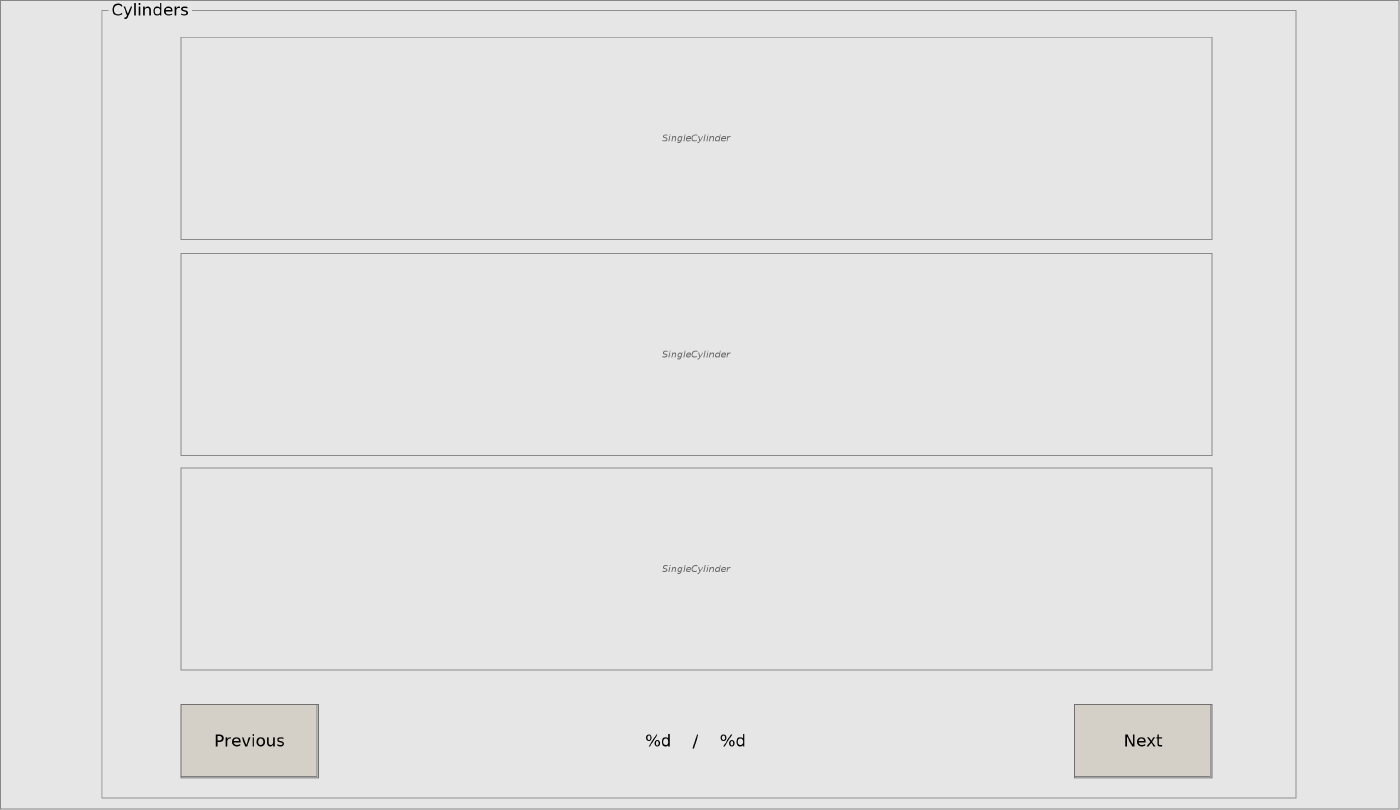
VISUALIZATION PageManualCylinders  // 1520x880
VAR_IN_OUT
	btnPrevious			: BOOL;
	btnNext				: BOOL;
	bPreviousInvisible	: BOOL;
	bNextInvisible		: BOOL;
	stCylinderEmpty		: ARRAY[1..3] OF BOOL;
	stCyliner			: ARRAY[1..3] OF ST_VisuCtrlCylinderFrame;
	iCylinderSelectedPageIndex	: USINT;
	iCylinderTotalPageIndex 	: USINT;
END_VAR
    GroupBox (110,3 1297x864), "Cylinders"
        Button (86,762 150x80), "Previous", invisible if: bPreviousInvisible
            tap btnPrevious
        Button (1056,762 150x80), "Next", invisible if: bNextInvisible
            tap btnNext
        Frame (86,37 1120x220), invisible if: stCylinderEmpty[1]
            shows SingleCylinder(stCylinder := stCyliner[1])
        Frame (86,272 1120x220), invisible if: stCylinderEmpty[2]
            shows SingleCylinder(stCylinder := stCyliner[2])
        Frame (86,505 1120x220), invisible if: stCylinderEmpty[3]
            shows SingleCylinder(stCylinder := stCyliner[3])
        Rectangle (580,777 130x50), "/"
        Rectangle (580,777 50x50), "%d", text variable: iCylinderSelectedPageIndex+1
        Rectangle (661,777 50x50), "%d", text variable: iCylinderTotalPageIndex+1
END_VISUALIZATION

(* stored: Version 1.1.0.1, ProductVersion 3.1.4024.12
   Visu PageManualCylinders: Id {ff9a9767-fe5b-4490-9b93-ff36f9b76073} *)
